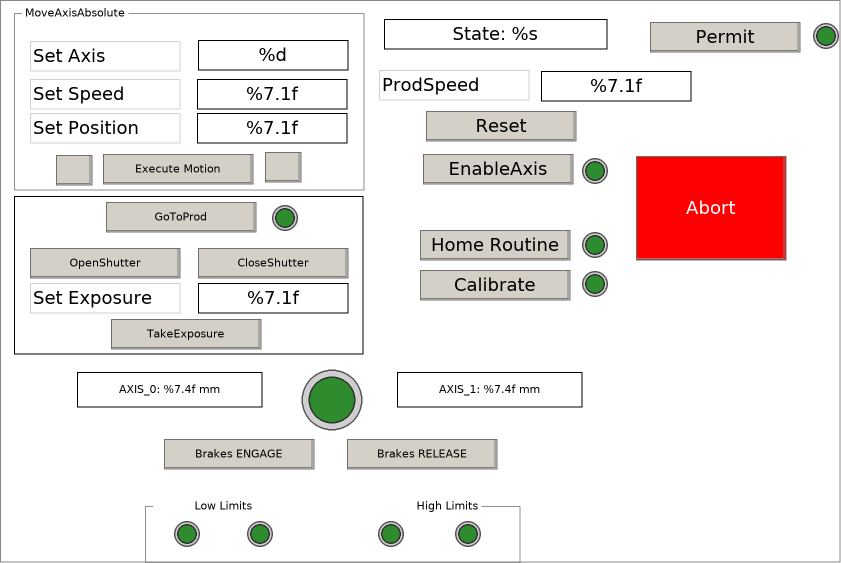
VISUALIZATION Visualization  // 841x563
    Rectangle (14,196 349x158)
    GroupBox (14,5 350x185), "MoveAxisAbsolute"
        Textfield (16,74 150x30), "Set Speed"
            OnMouseUp: write MAIN.inMoveAxisAbsolute.speed via Default, min 0, max 1667, format %7.1f
        Rectangle (183,74 150x30), "%7.1f", text variable: MAIN.inMoveAxisAbsolute.speed
        Textfield (16,108 150x30), "Set Position"
            OnMouseUp: write MAIN.inMoveAxisAbsolute.position via Default, min 0, max 751, format %7.1f
        Rectangle (183,108 150x30), "%7.1f", text variable: MAIN.inMoveAxisAbsolute.position
        Button (89,149 150x30), "Execute Motion"
            OnMouseUp: execute { MAIN.inMoveAxisAbsolute.dtime := MAIN.inMoveAxisAbsolute.dtime + 1; }
        Button (251,147 36x30)
            OnMouseUp: execute { MAIN.inMoveAxisAbsolute.position:=750.76; }
        Button (42,150 36x30)
            OnMouseUp: execute { MAIN.inMoveAxisAbsolute.position:=0; }
    Button (347,439 150x30), "Brakes RELEASE"
        OnMouseDown: execute {
            MAIN.inChangeBrakeState.axisIndex := 0;
            MAIN.inChangeBrakeState.state := FALSE;
            MAIN.inChangeBrakeState.dtime := MAIN.inChangeBrakeState.dtime + 1;
        }
        OnMouseUp: execute {
            MAIN.inChangeBrakeState.axisIndex := 1;
            MAIN.inChangeBrakeState.state := FALSE;
            MAIN.inChangeBrakeState.dtime := MAIN.inChangeBrakeState.dtime + 1;
        }
    Lamp1 (297,365 70x70), variable: (MAIN.stAxis[0].bBrake and MAIN.stAxis[1].bBrake), style: Lamp-Lamp1-Green
    Rectangle (77,372 185x35), "AXIS_0: %7.4f mm", text variable: MAIN.stAxis[0].axisRef.NcToPlc.ActPos
    Rectangle (397,372 185x35), "AXIS_1: %7.4f mm", text variable: MAIN.stAxis[1].axisRef.NcToPlc.ActPos
    Button (426,111 150x30), "Reset"
        OnMouseUp: execute { MAIN.inReset.dtime := MAIN.inReset.dtime + 1; }
    Button (636,156 150x104), "Abort"
        OnMouseUp: execute { MAIN.inReset.dtime := MAIN.inReset.dtime + 1; }
    Rectangle (384,19 223x30), "State: %s", text variable: MAIN.outShutterStatus.smState
    Button (420,230 150x30), "Home Routine"
        OnMouseUp: execute { MAIN.inHomeAxis.dtime := MAIN.inHomeAxis.dtime + 1; }
    Textfield (30,41 150x30), "Set Axis"
        OnMouseUp: write MAIN.inMoveAxisAbsolute.axisIndex via Default, min 0, max 1, format %b
    Rectangle (198,40 150x30), "%d", text variable: MAIN.inMoveAxisAbsolute.axisIndex
    Lamp1 (580,230 30x30), variable: MAIN.stAxis[0].axisRef.Status.Homed and MAIN.stAxis[1].axisRef.Status.Homed, style: Lamp-Lamp1-Green
    Button (420,270 150x30), "Calibrate"
        OnMouseUp: execute { MAIN.inCalibrate.dtime := MAIN.inCalibrate.dtime + 1; }
    Button (164,439 150x30), "Brakes ENGAGE"
        OnMouseDown: execute {
            MAIN.inChangeBrakeState.axisIndex := 0;
            MAIN.inChangeBrakeState.state := TRUE;
            MAIN.inChangeBrakeState.dtime := MAIN.inChangeBrakeState.dtime + 1;
        }
        OnMouseUp: execute {
            MAIN.inChangeBrakeState.axisIndex := 1;
            MAIN.inChangeBrakeState.state := TRUE;
            MAIN.inChangeBrakeState.dtime := MAIN.inChangeBrakeState.dtime + 1;
        }
    Button (650,22 150x30), "Permit"
        OnMouseDown: execute { MAIN.bAuxElxPermit := NOT MAIN.bAuxElxPermit; }
    Lamp1 (811,21 30x30), variable: MAIN.bAuxElxPermit, style: Lamp-Lamp1-Green
    Button (423,154 150x30), "EnableAxis"
        OnMouseUp: execute { MAIN.inEnableAllAxes.dtime := MAIN.inEnableAllAxes.dtime + 1; }
    Button (106,202 150x30), "GoToProd"
        OnMouseUp: execute { MAIN.inGoToProd.dtime := MAIN.inGoToProd.dtime + 1; }
    Button (30,248 150x30), "OpenShutter"
        OnMouseUp: execute { MAIN.inOpenShutter.dtime := MAIN.inOpenShutter.dtime + 1; }
    Button (198,248 150x30), "CloseShutter"
        OnMouseUp: execute { MAIN.inCloseShutter.dtime := MAIN.inCloseShutter.dtime + 1; }
    Button (111,319 150x30), "TakeExposure"
        OnMouseUp: execute { MAIN.inTakeExposure.dtime := MAIN.inTakeExposure.dtime + 1; }
    Rectangle (541,71 150x30), "%7.1f", text variable: MAIN.inReset.speed
    Textfield (379,70 150x30), "ProdSpeed"
        OnMouseUp: write MAIN.inReset.speed via Default, min 0, max 1667, format %7.1f
    Textfield (30,283 150x30), "Set Exposure"
        OnMouseUp: write MAIN.inTakeExposure.exposureTime via Default, min 100, format %7.1f
    Rectangle (198,283 150x30), "%7.1f", text variable: MAIN.inTakeExposure.exposureTime
    Lamp1 (580,269 30x30), variable: MAIN.stAxis[0].bIsCalibrated and MAIN.stAxis[1].bIsCalibrated;, style: Lamp-Lamp1-Green
    Lamp1 (580,156 30x30), variable: MAIN.outShutterStatus.axis[0].enabled and MAIN.outShutterStatus.axis[1].enabled;, style: Lamp-Lamp1-Green
    Lamp1 (172,519 30x30), variable: MAIN.stAxis[0].bLimitHome;, style: Lamp-Lamp1-Green
    Lamp1 (245,519 30x30), variable: MAIN.stAxis[1].bLimitDeployed;, style: Lamp-Lamp1-Green
    Lamp1 (376,519 30x30), variable: MAIN.stAxis[0].bLimitDeployed;, style: Lamp-Lamp1-Green
    Lamp1 (453,519 30x30), variable: MAIN.stAxis[1].bLimitHome;, style: Lamp-Lamp1-Green
    GroupBox (145,498 375x65), "Low Limits High Limits"
    Lamp1 (270,203 30x30), variable: MAIN.fbShutterSM.fbEnabled.bShutterReady;, style: Lamp-Lamp1-Green
END_VISUALIZATION

(* stored: Version 1.1.0.1, ProductVersion 3.1.4024.4
   Visu Visualization: Id {f582b681-f1ff-4fd0-9241-dc5537cf3bfd} *)
